
// ===== library types =====

FUNCTION_BLOCK "TASK1"   // FB1, LAD
{ S7_Optimized_Access := 'TRUE' }
VERSION : 0.1
   VAR_INPUT
      Start : Bool;
      Stop : Bool;
      reset : Bool;
      "Timer" : DInt;   // value in milliseconds
      "max temperature" : Real;   // max temperature you want in the tank
      "min temperature" : Real;   // min temperature you want in the tank
      "reset temp" : Real;   // to reset the temperature
      "any value" : Real;
      manual : Bool;
   END_VAR
   VAR_OUTPUT
      Output_1 : Bool;
   END_VAR
   VAR_IN_OUT
      Run : Bool;   // process is working
      Heater : Bool;
      "max limit" : Bool;
      "min limit" : Bool;
      Temperature : Real;
   END_VAR
   VAR
      Ton : Bool;
      Toff : Bool;   // reset the timer
      IEC_Timer_0_Instance_1 : TON_TIME;
   END_VAR
BEGIN

REGION Network 1: control operarion
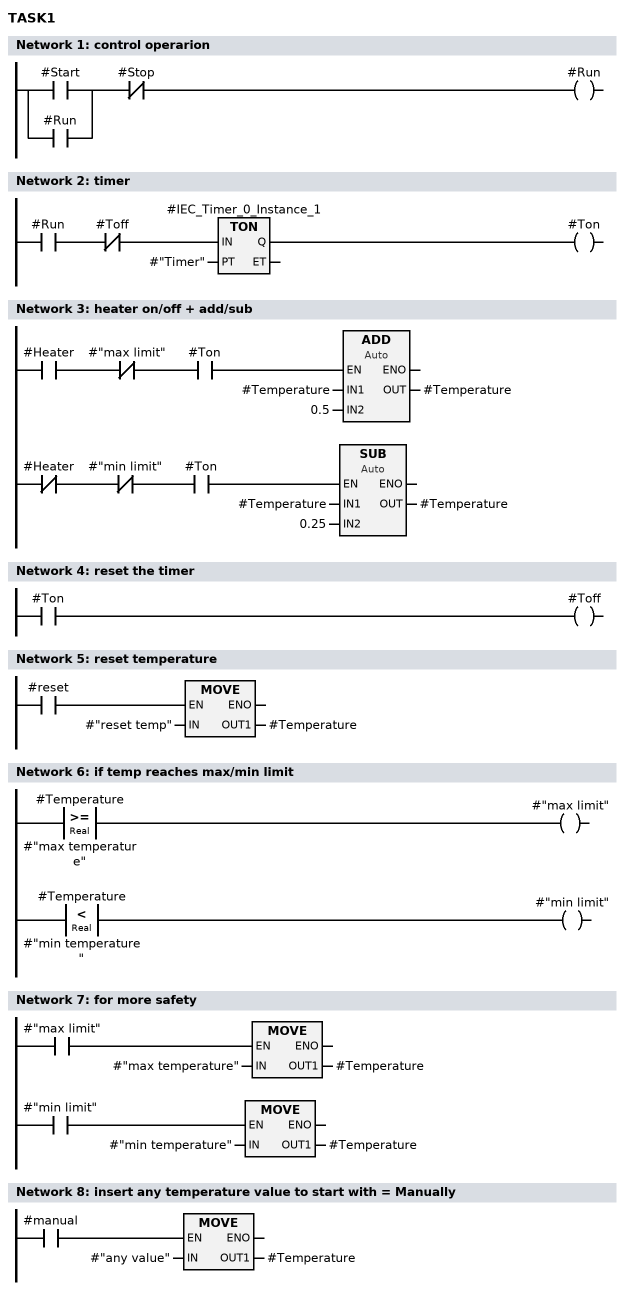
   RUNG wire#powerrail
      Contact( #Start )
      wire#w1
      I_Contact( #Stop )
      Coil( #Run )
   END_RUNG
   RUNG wire#powerrail
      Contact( #Run )
   END_RUNG wire#w1
   // the same network as SCL:
   #Run := (#Start OR #Run) AND NOT #Stop;
END_REGION

REGION Network 2: timer
   #IEC_Timer_0_Instance_1(IN := #Run AND NOT #Toff, PT := #"Timer");   // TON
   #Ton := #IEC_Timer_0_Instance_1.Q;
END_REGION

REGION Network 3: heater on/off + add/sub
   RUNG wire#powerrail
      Contact( #Heater )
      I_Contact( #"max limit" )
      Contact( #Ton )
      Add(in1 := #Temperature, in2 := 0.5, out => #Temperature)
   END_RUNG
   RUNG wire#powerrail
      I_Contact( #Heater )
      I_Contact( #"min limit" )
      Contact( #Ton )
      Sub(in1 := #Temperature, in2 := 0.25, out => #Temperature)
   END_RUNG
   // the same network as SCL:
   IF #Heater AND NOT #"max limit" AND #Ton THEN #Temperature := #Temperature + 0.5; END_IF;
   IF NOT #Heater AND NOT #"min limit" AND #Ton THEN #Temperature := #Temperature - 0.25; END_IF;
END_REGION

REGION Network 4: reset the timer
   RUNG wire#powerrail
      Contact( #Ton )
      Coil( #Toff )
   END_RUNG
   // the same network as SCL:
   #Toff := #Ton;
END_REGION

REGION Network 5: reset temperature
   RUNG wire#powerrail
      Contact( #reset )
      Move(in := #"reset temp", out1 => #Temperature)
   END_RUNG
   // the same network as SCL:
   IF #reset THEN #Temperature := #"reset temp"; END_IF;
END_REGION

REGION Network 6: if temp reaches max/min limit
   RUNG wire#powerrail
      { S7_Templates := "SrcType := Real" } GE_Contact(in1 := #Temperature, in2 := #"max temperature")
      Coil( #"max limit" )
   END_RUNG
   RUNG wire#powerrail
      { S7_Templates := "SrcType := Real" } LT_Contact(in1 := #Temperature, in2 := #"min temperature")
      Coil( #"min limit" )
   END_RUNG
   // the same network as SCL:
   #"max limit" := #Temperature >= #"max temperature";
   #"min limit" := #Temperature < #"min temperature";
END_REGION

REGION Network 7: for more safety
   RUNG wire#powerrail
      Contact( #"max limit" )
      Move(in := #"max temperature", out1 => #Temperature)
   END_RUNG
   RUNG wire#powerrail
      Contact( #"min limit" )
      Move(in := #"min temperature", out1 => #Temperature)
   END_RUNG
   // the same network as SCL:
   IF #"max limit" THEN #Temperature := #"max temperature"; END_IF;
   IF #"min limit" THEN #Temperature := #"min temperature"; END_IF;
END_REGION

REGION Network 8: insert any temperature value to start with = Manually
   RUNG wire#powerrail
      Contact( #manual )
      Move(in := #"any value", out1 => #Temperature)
   END_RUNG
   // the same network as SCL:
   IF #manual THEN #Temperature := #"any value"; END_IF;
END_REGION
END_FUNCTION_BLOCK